// Block: CoilHandling_PERS

DATA_BLOCK CoilHandling_PERS
VERSION : 0.1
   NON_RETAIN
   VAR
      PersistentValues : CoilHandling_Persistent;
   END_VAR

BEGIN
   // No initialization required
END_DATA_BLOCK
